// TIA Portal V16 export
// export: Created 2021-04-11T09:51:32.8023181Z, ExportSetting WithDefaults, DisplayName Totally Integrated Automation Portal, DisplayVersion V16, DisplayName TIA Portal Version Control Interface, DisplayVersion V16, DisplayName TIA Portal Openness, DisplayVersion V16, DisplayName STEP 7 Professional, DisplayVersion V16, DisplayName STEP 7 Safety, DisplayVersion V16, DisplayName WinCC Unified SCADA Engineering System, DisplayVersion V16
FUNCTION "findSum" : Void   // FC8, LAD
{ S7_Optimized_Access := 'TRUE' }
VERSION : 0.1
// stored: AutoNumber true, IsIECCheckEnabled false, SetENOAutomatically false, UDAEnableTagReadback false
   VAR_INPUT
      arrWeight : Array[0..12] of Real;
      arrBitMask : Array[0..12] of Bool;
   END_VAR
   VAR_IN_OUT
      tmpSum : Real;
   END_VAR
BEGIN

REGION Network 1 (SCL)
   #tmpSum := #arrWeight[0] * BOOL_TO_INT(#arrBitMask[0]) +
   #arrWeight[1] * BOOL_TO_INT(#arrBitMask[1])+
   #arrWeight[2] * BOOL_TO_INT(#arrBitMask[2]) +
   #arrWeight[3] * BOOL_TO_INT(#arrBitMask[3]) +
   #arrWeight[4] * BOOL_TO_INT(#arrBitMask[4]) +
   #arrWeight[5] * BOOL_TO_INT(#arrBitMask[5]) +
   #arrWeight[6] * BOOL_TO_INT(#arrBitMask[6]) +
   #arrWeight[7] * BOOL_TO_INT(#arrBitMask[7]) +
   #arrWeight[8] * BOOL_TO_INT(#arrBitMask[8]) +
   #arrWeight[9] * BOOL_TO_INT(#arrBitMask[9]) +
   #arrWeight[10] * BOOL_TO_INT(#arrBitMask[10]) +
   #arrWeight[11] * BOOL_TO_INT(#arrBitMask[11]) +
   #arrWeight[12] * BOOL_TO_INT(#arrBitMask[12]);
END_REGION
END_FUNCTION
